FUNCTION_BLOCK EL3111
VAR
	_io : EL3xx1_Data;
	{attribute addProperty Name "WcState"}
	_wcState : WcStateInputToggle;
	{attribute addProperty Name "Info data"}
	_infoData : InfoDataAds;
END_VAR

PROPERTY IO : REFERENCE TO EL3xx1_Data
GET
IO REF= _io;
END_GET
END_PROPERTY

PROPERTY WcState : REFERENCE TO WcStateInputToggle
GET
WcState REF= _wcState;
END_GET
END_PROPERTY

END_FUNCTION_BLOCK

(* stored: Version 1.1.0.1, ProductVersion 3.1.4024.9
   POU EL3111: Id {c067e485-88bb-02ba-0130-7a53155b4b6a}, SpecialFunc None
   Property IO: Id {13fd6def-e610-0b2d-28f6-9153d117042c}
   Get Get: Id {6821fffd-0a2a-0e94-30a8-a5a71eacb4bb}
   Property WcState: Id {15f54d4a-c185-000b-1d74-21422778b528}
   Get Get: Id {529e3607-52e2-046b-1770-bd180034b1e7} *)
